// TwinCAT 3 PLC project Variablenspeicher
// ProgramVersion: 3.1.4022.0
// libraries:
//   Tc2_Standard, * (Beckhoff Automation GmbH)
//   Tc2_System, * (Beckhoff Automation GmbH)
//   Tc3_Module, * (Beckhoff Automation GmbH)
// project tree:
//   GVLs/ vars.TcGVL
//   / PlcTask.TcTTO
//   POUs/ MAIN.TcPOU
// (motion and I/O tree: see PLC project shutdown)
// real-time tasks:
//   TASK Plc_Task: cycle T#10ms, priority 20, ADS port 350
//   TASK IrSensor_Task: cycle T#5ms, priority 9, ADS port 351
//   TASK UDP_Task: cycle T#10ms, priority 10, ADS port 354
//   TASK Regler_Task: cycle T#50000us, priority 1, ADS port 352
// variable links:
//   Variablenspeicher/Variablenspeicher Instance <-> TcCOM Objects/Object1 (Gewerk3_Simulinkmodell_2017_10_09_Twincat)
//     PlcTask Inputs/vars.fromMatlab_theta <-> Output/v_theta
//     PlcTask Inputs/vars.fromMatlab_velocityX <-> Output/v_x
//     PlcTask Inputs/vars.fromMatlab_velocityY <-> Output/v_y
//   Variablenspeicher/Variablenspeicher Instance <-> velocityConverterToMotors/velocityConverterToMotors_Obj
//     PlcTask Outputs/MAIN.theta <-> Inputs/theta
//     PlcTask Outputs/MAIN.velocityX <-> Inputs/velocityX
//     PlcTask Outputs/MAIN.velocityY <-> Inputs/velocityY

CONFIGURATION Variablenspeicher
    RESOURCE PLC ON TwinCAT3
        TASK PlcTask(INTERVAL := T#10ms, PRIORITY := 20);
        PROGRAM MAIN WITH PlcTask : MAIN;
    END_RESOURCE
END_CONFIGURATION

// ---- GVLs/vars.TcGVL
{attribute 'qualified_only'}
VAR_GLOBAL
	udp_x	: LREAL := 2000;
	udp_y	: LREAL := 1400;
	udp_theta : LREAL := 1.4;
	
	fromMatlab_velocityX AT%I* : LREAL;
	fromMatlab_velocityY AT%I*: LREAL;
	fromMatlab_theta AT%I*: LREAL;
	
END_VAR

// ---- POUs/MAIN.TcPOU
PROGRAM MAIN
VAR
	velocityX AT%Q* : LREAL;
	velocityY AT%Q* : LREAL;
	theta AT%Q* : LREAL;
END_VAR

velocityX := vars.fromMatlab_velocityX;
velocityY := vars.fromMatlab_velocityY;
theta := vars.fromMatlab_theta;

END_PROGRAM
